// TIA Portal V16 export
// export: Created 2022-07-21T09:35:16.2754695Z, ExportSetting WithDefaults, DisplayName Totally Integrated Automation Portal, DisplayVersion V16 Update 4, DisplayName TIA Portal Version Control Interface, DisplayVersion V16 Update 2, DisplayName TIA Portal Openness, DisplayVersion V16 Update 4, DisplayName SINAMICS Startdrive Advanced, DisplayVersion V16 Update 5, DisplayName SINAMICS Startdrive G130, G150, S120, S150, SINAMICS MV, S210, DisplayVersion V16 Update 5, DisplayName SINAMICS Startdrive G110M, G120, G120C, G120D, G120P, G115D, DisplayVersion V16 Update 5, DisplayName STEP 7 Professional, DisplayVersion V16 Update 4, DisplayName STEP 7 Safety, DisplayVersion V16, DisplayName WinCC Advanced, DisplayVersion V16 Update 4
FUNCTION_BLOCK "fbMessageHandlingRate"   // FB87, LAD
TITLE = Camera handling / Obsługa kamery
{ S7_Optimized_Access := 'TRUE' }
VERSION : 0.1
// stored: AutoNumber true, IsIECCheckEnabled true, IsRetainMemResEnabled false, MemoryReserve 100, SetENOAutomatically false, UDAEnableTagReadback false
   VAR_INPUT
      inEnable { ExternalAccessible := 'False'; ExternalVisible := 'False'; ExternalWritable := 'False'} : Bool;   // Zezwolenie / Enable
      inFbOk { ExternalAccessible := 'False'; ExternalVisible := 'False'; ExternalWritable := 'False'} : Bool;   // Odczyt ok / Read ok
      inFbNotOk { ExternalAccessible := 'False'; ExternalVisible := 'False'; ExternalWritable := 'False'} : Bool;   // Odczyt nok / Read nok
      inRateWarning { ExternalAccessible := 'False'; ExternalVisible := 'False'; ExternalWritable := 'False'} : Real;   // Wskaznik dla ostrzeżenia / Rate warning
      inRateError { ExternalAccessible := 'False'; ExternalVisible := 'False'; ExternalWritable := 'False'} : Real;   // Wskaznik dla błędu / Rate error
      inAmountTillMessage { ExternalAccessible := 'False'; ExternalVisible := 'False'; ExternalWritable := 'False'} : USInt;   // Ilość błędnych odczytów do ustawienia błędu / Amount of bad reads till error
      inResetMessages { ExternalAccessible := 'False'; ExternalVisible := 'False'; ExternalWritable := 'False'} : Bool;   // Sygnał resetu / Reset
   END_VAR
   VAR_OUTPUT
      ouMsgWarning { ExternalAccessible := 'False'; ExternalVisible := 'False'; ExternalWritable := 'False'} : Bool;   // Ostrzeżenie / Warning
      ouMsgError { ExternalAccessible := 'False'; ExternalVisible := 'False'; ExternalWritable := 'False'} : Bool;   // Błąd / Error
   END_VAR
   VAR
      sCntOkayWarning { ExternalAccessible := 'False'; ExternalVisible := 'False'; ExternalWritable := 'False'} : UDInt;
      sCntNotOkayWarning { ExternalAccessible := 'False'; ExternalVisible := 'False'; ExternalWritable := 'False'} : USInt;
      sCntOkayError { ExternalAccessible := 'False'; ExternalVisible := 'False'; ExternalWritable := 'False'} : UDInt;
      sCntNotOkayError { ExternalAccessible := 'False'; ExternalVisible := 'False'; ExternalWritable := 'False'} : USInt;
      sMessageWarning { ExternalAccessible := 'False'; ExternalVisible := 'False'; ExternalWritable := 'False'; S7_SetPoint := 'True'} : "fbMessageHandlingDelayed";
      sMessageError { ExternalAccessible := 'False'; ExternalVisible := 'False'; ExternalWritable := 'False'; S7_SetPoint := 'True'} : "fbMessageHandlingDelayed";
   END_VAR
   VAR_TEMP
      tLimitWarning : UDInt;
      tLimitError : UDInt;
      tStatusWarning : USInt;
      tStatusError : USInt;
   END_VAR
BEGIN

REGION Network 1 (SCL): Counters / Liczniki

   // Calculate limits
   #tLimitWarning := ROUND_UDINT(100.0 / (100.0 - #inRateWarning));
   #tLimitError   := ROUND_UDINT(100.0 / (100.0 - #inRateError));

   // Count not okay
   IF #inFbNotOk THEN
     #sCntNotOkayError += 1;
     #sCntNotOkayWarning += 1;
   END_IF;

   // Count okay
   IF #inFbOk THEN
     // counter for error
     #sCntOkayError += 1;
     IF #sCntOkayError >= #tLimitError THEN
       #sCntOkayError := 0;
       IF #sCntNotOkayError > 0 THEN
         #sCntNotOkayError -= 1;
       END_IF;
     END_IF;

     // counter for warning
     #sCntOkayWarning += 1;
     IF #sCntOkayWarning >= #tLimitWarning THEN
       #sCntOkayWarning := 0;
       IF #sCntNotOkayWarning > 0 THEN
         #sCntNotOkayWarning -= 1;
       END_IF;
     END_IF;
   END_IF;

   // Clear counter on error
   IF #ouMsgError
       OR #inAmountTillMessage <= 0
       OR #inRateError <= 0
   THEN
     // Counter for error
     #sCntOkayError := 0;
     #sCntNotOkayError := 0;

     // Counter for warning
     #sCntOkayWarning := 0;
     #sCntNotOkayWarning := 0;
   END_IF;
END_REGION

REGION Network 2: Error handling / Obsługa błędów
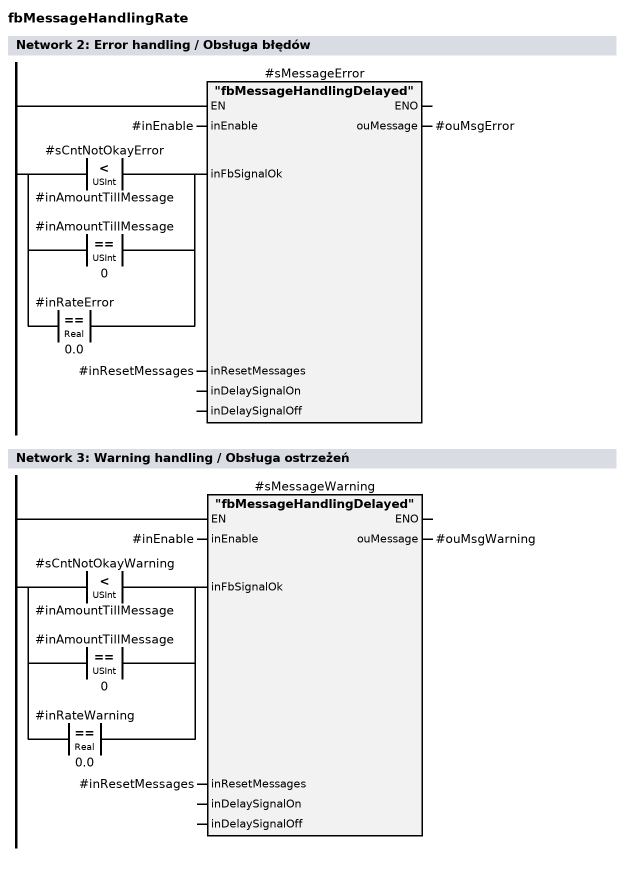
   RUNG wire#powerrail
      #sMessageError(inFbSignalOk := wire#w1, inEnable := #inEnable, inResetMessages := #inResetMessages, inDelaySignalOn :=, inDelaySignalOff :=, ouMessage => #ouMsgError)
   END_RUNG
   RUNG wire#powerrail
      { S7_Templates := "SrcType := USInt" } LT_Contact(in1 := #sCntNotOkayError, in2 := #inAmountTillMessage)
   END_RUNG wire#w1
   RUNG wire#powerrail
      { S7_Templates := "SrcType := USInt" } EQ_Contact(in1 := #inAmountTillMessage, in2 := 0)
   END_RUNG wire#w1
   RUNG wire#powerrail
      { S7_Templates := "SrcType := Real" } EQ_Contact(in1 := #inRateError, in2 := 0.0)
   END_RUNG wire#w1
   // the same network as SCL:
   #sMessageError(inEnable := #inEnable,   // "fbMessageHandlingDelayed"
                  inFbSignalOk := (#sCntNotOkayError < #inAmountTillMessage) OR (#inAmountTillMessage = 0) OR (#inRateError = 0.0),
                  inResetMessages := #inResetMessages,
                  ouMessage => #ouMsgError);
END_REGION

REGION Network 3: Warning handling / Obsługa ostrzeżeń
   RUNG wire#powerrail
      #sMessageWarning(inFbSignalOk := wire#w1, inEnable := #inEnable, inResetMessages := #inResetMessages, inDelaySignalOn :=, inDelaySignalOff :=, ouMessage => #ouMsgWarning)
   END_RUNG
   RUNG wire#powerrail
      { S7_Templates := "SrcType := USInt" } LT_Contact(in1 := #sCntNotOkayWarning, in2 := #inAmountTillMessage)
   END_RUNG wire#w1
   RUNG wire#powerrail
      { S7_Templates := "SrcType := USInt" } EQ_Contact(in1 := #inAmountTillMessage, in2 := 0)
   END_RUNG wire#w1
   RUNG wire#powerrail
      { S7_Templates := "SrcType := Real" } EQ_Contact(in1 := #inRateWarning, in2 := 0.0)
   END_RUNG wire#w1
   // the same network as SCL:
   #sMessageWarning(inEnable := #inEnable,   // "fbMessageHandlingDelayed"
                    inFbSignalOk := (#sCntNotOkayWarning < #inAmountTillMessage) OR (#inAmountTillMessage = 0) OR (#inRateWarning = 0.0),
                    inResetMessages := #inResetMessages,
                    ouMessage => #ouMsgWarning);
END_REGION
END_FUNCTION_BLOCK
